FUNCTION_BLOCK SS3_ifb_ps_Vibrator (* Composite FB wrapping other FBs *)
  (* Standard: 61499-2 *)
  (* Version 1.0, 2025-05-16, PS_Transformer_for_Unknown *)
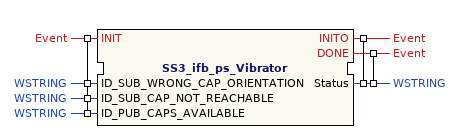
  EVENT_INPUT
    INIT WITH ID_SUB_WRONG_CAP_ORIENTATION, ID_SUB_CAP_NOT_REACHABLE, ID_PUB_CAPS_AVAILABLE; (* Initialization Request *)
  END_EVENT
  EVENT_OUTPUT
    INITO WITH Status; (* Initialization Confirm *)
    DONE WITH Status; (* Execution Confirmation *)
  END_EVENT
  VAR_INPUT
    ID_SUB_WRONG_CAP_ORIENTATION : WSTRING;
    ID_SUB_CAP_NOT_REACHABLE : WSTRING;
    ID_PUB_CAPS_AVAILABLE : WSTRING;
  END_VAR
  VAR_OUTPUT
    Status : WSTRING; (* Output event qualifier *)
  END_VAR
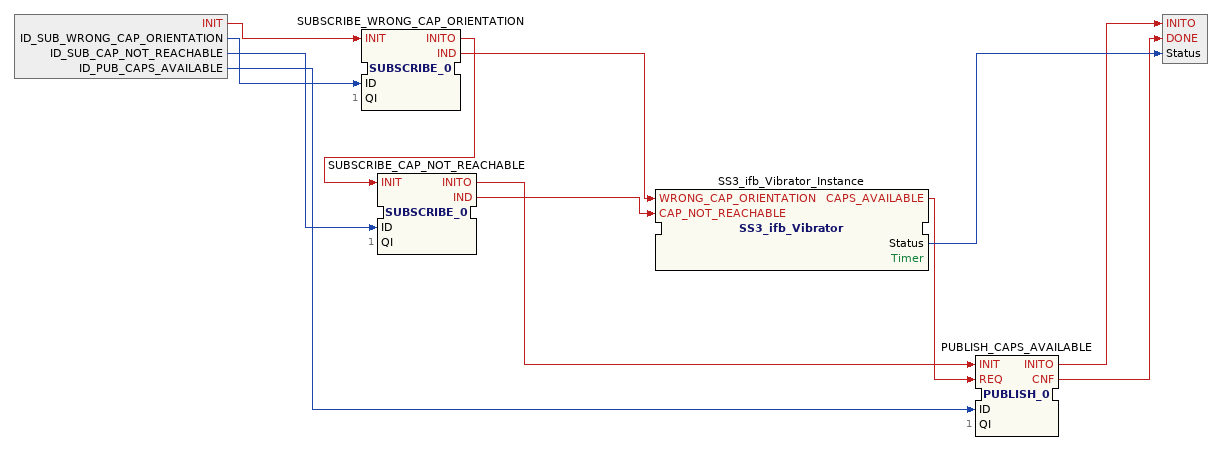
  FBS
    SS3_ifb_Vibrator_Instance : SS3_ifb_Vibrator;
    SUBSCRIBE_WRONG_CAP_ORIENTATION : SUBSCRIBE_0(QI := 1);
    SUBSCRIBE_CAP_NOT_REACHABLE : SUBSCRIBE_0(QI := 1);
    PUBLISH_CAPS_AVAILABLE : PUBLISH_0(QI := 1);
  END_FBS
  EVENT_CONNECTIONS
    INIT TO SUBSCRIBE_WRONG_CAP_ORIENTATION.INIT;
    SUBSCRIBE_WRONG_CAP_ORIENTATION.INITO TO SUBSCRIBE_CAP_NOT_REACHABLE.INIT;
    SUBSCRIBE_CAP_NOT_REACHABLE.INITO TO PUBLISH_CAPS_AVAILABLE.INIT;
    PUBLISH_CAPS_AVAILABLE.INITO TO INITO;
    SUBSCRIBE_WRONG_CAP_ORIENTATION.IND TO SS3_ifb_Vibrator_Instance.WRONG_CAP_ORIENTATION;
    SUBSCRIBE_CAP_NOT_REACHABLE.IND TO SS3_ifb_Vibrator_Instance.CAP_NOT_REACHABLE;
    SS3_ifb_Vibrator_Instance.CAPS_AVAILABLE TO PUBLISH_CAPS_AVAILABLE.REQ;
    PUBLISH_CAPS_AVAILABLE.CNF TO DONE;
  END_CONNECTIONS
  DATA_CONNECTIONS
    ID_SUB_WRONG_CAP_ORIENTATION TO SUBSCRIBE_WRONG_CAP_ORIENTATION.ID;
    ID_SUB_CAP_NOT_REACHABLE TO SUBSCRIBE_CAP_NOT_REACHABLE.ID;
    ID_PUB_CAPS_AVAILABLE TO PUBLISH_CAPS_AVAILABLE.ID;
    SS3_ifb_Vibrator_Instance.Status TO Status;
  END_CONNECTIONS
END_FUNCTION_BLOCK
